Yaskawa INFORM job: CYLINDER2.JBI

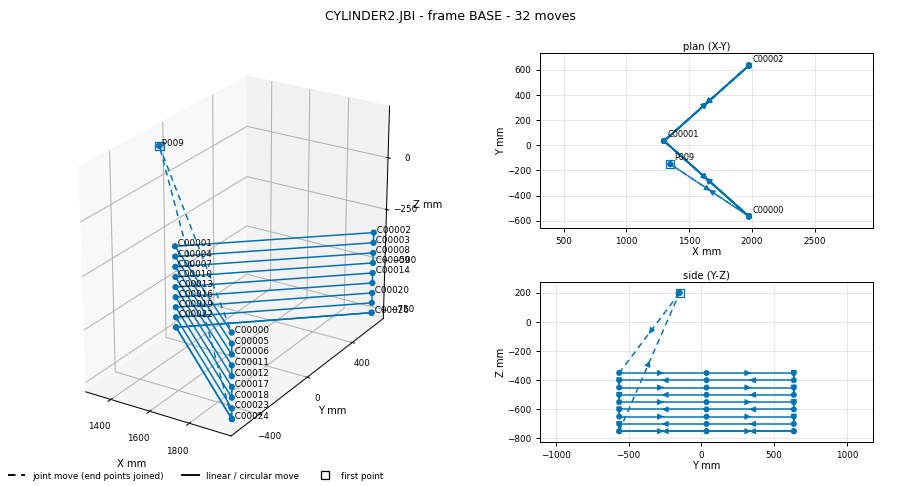
[picture p0: tool path of CYLINDER2.JBI in frame BASE, 32 of 32 moves have a stored position in this frame; points joined in program order, loops and branches not executed]
/JOB
//NAME CYLINDER2
//POS
///NPOS 30,0,30,1,0,1
///TOOL 0
///POSTYPE BASE
///RECTAN
///RCONF 0,0,0,0,0,0,0,0,0,0,0,0,0,0,0,0,0,0,0,0,0,0,0,0
C00000=1975.005,-565.000,-350.000,-180.0000,-90.0000,90.0000
C00001=1300.000,35.000,-350.000,-180.0000,-90.0000,0.0000
C00002=1975.000,635.000,-350.000,-180.0000,-90.0000,-90.0000
C00003=1975.000,635.000,-400.000,-180.0000,-90.0000,-90.0000
C00004=1300.000,35.000,-400.000,-180.0000,-90.0000,0.0000
C00005=1975.000,-565.000,-400.000,-180.0000,-90.0000,90.0000
C00006=1975.000,-565.000,-450.000,-180.0000,-90.0000,90.0000
C00007=1300.000,35.000,-450.000,-180.0000,-90.0000,0.0000
C00008=1975.000,635.000,-450.000,-180.0000,-90.0000,-90.0000
C00009=1975.000,635.000,-500.000,-180.0000,-90.0000,-90.0000
C00010=1300.000,35.000,-500.000,-180.0000,-90.0000,0.0000
C00011=1975.000,-565.000,-500.000,-180.0000,-90.0000,90.0000
C00012=1975.000,-565.000,-550.000,-180.0000,-90.0000,90.0000
C00013=1300.000,35.000,-550.000,-180.0000,-90.0000,0.0000
C00014=1975.000,635.000,-550.000,-180.0000,-90.0000,-90.0000
C00015=1975.000,635.000,-600.000,-180.0000,-90.0000,-90.0000
C00016=1300.000,35.000,-600.000,-180.0000,-90.0000,0.0000
C00017=1975.000,-565.000,-600.000,-180.0000,-90.0000,90.0000
C00018=1975.000,-565.000,-650.000,-180.0000,-90.0000,90.0000
C00019=1300.000,35.000,-650.000,-180.0000,-90.0000,0.0000
C00020=1975.000,635.000,-650.000,-180.0000,-90.0000,-90.0000
C00021=1975.000,635.000,-700.000,-180.0000,-90.0000,-90.0000
C00022=1300.000,35.000,-700.000,-180.0000,-90.0000,0.0000
C00023=1975.000,-565.000,-700.000,-180.0000,-90.0000,90.0000
C00024=1975.000,-565.000,-750.000,-180.0000,-90.0000,90.0000
C00025=1300.000,35.000,-750.000,-180.0000,-90.0000,0.0000
C00026=1975.000,635.000,-750.000,-180.0000,-90.0000,-90.0000
C00027=1975.000,635.000,-750.000,180.0000,-70.0000,-90.0000
C00028=1300.000,35.000,-750.000,-180.0000,-70.0000,0.0000
C00029=1975.000,-565.000,-750.000,180.0000,-70.0000,90.0000
///POSTYPE PULSE
///PULSE
EC00000=0
EC00001=0
EC00002=0
EC00003=0
EC00004=0
EC00005=0
EC00006=0
EC00007=0
EC00008=0
EC00009=0
EC00010=0
EC00011=0
EC00012=0
EC00013=0
EC00014=0
EC00015=0
EC00016=0
EC00017=0
EC00018=0
EC00019=0
EC00020=0
EC00021=0
EC00022=0
EC00023=0
EC00024=0
EC00025=0
EC00026=0
EC00027=0
EC00028=0
EC00029=0
///POSTYPE BASE
///RECTAN
P00009=1350.000,-150.000,200.000,-180.0000,-45.0000,0.0000
///POSTYPE PULSE
///PULSE
EX00000=0
//INST
///DATE 2023/02/13 19:51
///ATTR SC,RW,RJ
////FRAME BASE
///GROUP1 RB1,ST1
NOP
MOVJ P009 EX000 VJ=15.00
MOVJ C00000 EC00000 VJ=15.00
CALL JOB:SPYON
MOVC C00001 EC00001 V=150.0
MOVC C00002 EC00002 V=150.0
MOVL C00003 EC00003 V=150.0
MOVC C00004 EC00004 V=150.0
MOVC C00005 EC00005 V=150.0
MOVL C00006 EC00006 V=150.0
MOVC C00007 EC00007 V=150.0
MOVC C00008 EC00008 V=150.0
MOVL C00009 EC00009 V=150.0
MOVC C00010 EC00010 V=150.0
MOVC C00011 EC00011 V=150.0
MOVL C00012 EC00012 V=150.0
MOVC C00013 EC00013 V=150.0
MOVC C00014 EC00014 V=150.0
MOVL C00015 EC00015 V=150.0
MOVC C00016 EC00016 V=150.0
MOVC C00017 EC00017 V=150.0
MOVL C00018 EC00018 V=150.0
MOVC C00019 EC00019 V=150.0
MOVC C00020 EC00020 V=150.0
MOVL C00021 EC00021 V=150.0
MOVC C00022 EC00022 V=150.0
MOVC C00023 EC00023 V=150.0
MOVL C00024 EC00024 V=150.0
MOVC C00025 EC00025 V=150.0
MOVC C00026 EC00026 V=150.0
MOVL C00027 EC00027 V=150.0
MOVC C00028 EC00028 V=150.0
MOVC C00029 EC00029 V=150.0
CALL JOB:SPYOF
MOVJ P009 EX000 VJ=15.00
END
